PROGRAM MAIN

	VAR
		Seedra          : FB_Machine := (Name := 'SeedraMAIN');
		InitComplete    : BOOL;
		RebootSystem	: NT_Reboot;
	END_VAR

CyclicLogic();
//TESTS();

METHOD CyclicLogic
VAR_INPUT
END_VAR
IF NOT InitComplete THEN
    InitComplete := Initialize();
    RETURN;
END_IF

//Machine support HMI & Production Monitor


//Machine Cyclic Logic
Seedra.CyclicLogic();
END_METHOD

METHOD Initialize : BOOL
VAR_INPUT
END_VAR
//Top level machine initialization should happen here, in the main initialization method. Each subsequent "layer" of modules will be named within their respective "parent" intialize method
_AppInfo.KeepOutputsOnBP := TRUE;
Initialize := TRUE;
END_METHOD

END_PROGRAM

(* stored: Version 1.1.0.1, ProductVersion 3.1.4024.15
   POU MAIN: Id {0464503f-a0ee-0a19-098a-507ac5cd340b}, SpecialFunc None
   Method CyclicLogic: Id {85924404-3ac7-07ce-3884-239a0c5cad48}
   Method Initialize: Id {be8521cc-b0d4-05ce-0dc0-3bdba453ebf5} *)
